{attribute 'qualified_only'}
{attribute 'strict'}
TYPE E_MachineProfile :
(
    eProduction,    
    eManual         
);
END_TYPE

(* stored: Version 1.1.0.1, ProductVersion 3.1.4024.15
   DUT E_MachineProfile: Id {40400825-fd66-4322-b0cf-4871cdbc3d9c} *)
